// Mitsubishi GX Works2 project: GX W2 L2 Ex 3 DK c   PLC: FX3G

// global labels: Global1
VAR_GLOBAL
  iStart_PB AT X001 : BOOL;
  iStop_PB AT X002 : BOOL;
  bSystem_started : BOOL;
  oConveyer_Belt AT Y001 : BOOL;
END_VAR

// task Task_01 (event TRUE, interval 0, priority 31): POU_01

PROGRAM POU_01
VAR
  TON_2_OffTimer : TON;
  TON_1_OnTimer : TON;
END_VAR
(* structured ladder/FBD written out as ST: instructions are called as NAME(EN, inputs, outputs); _pN, _eN, _tN stand for wires *)
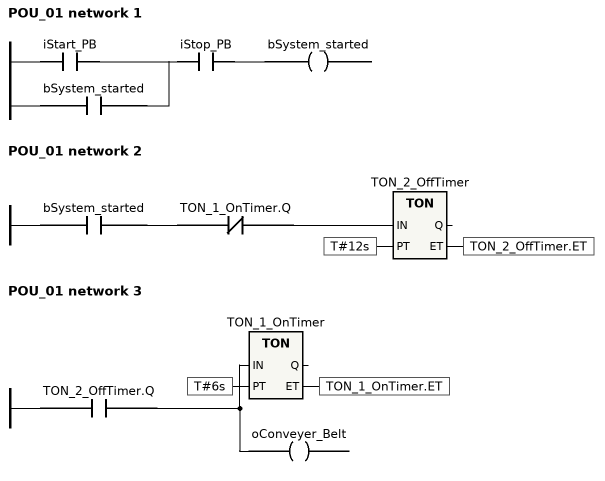
(* network 1 *)
bSystem_started := (iStart_PB OR bSystem_started) AND iStop_PB;
(* network 2 *)
TON_2_OffTimer(IN := bSystem_started AND NOT TON_1_OnTimer.Q, PT := T#12s, ET => TON_2_OffTimer.ET);
(* network 3 *)
TON_1_OnTimer(IN := TON_2_OffTimer.Q, PT := T#6s, ET => TON_1_OnTimer.ET);
oConveyer_Belt := TON_2_OffTimer.Q;
END_PROGRAM
